FUNCTION_BLOCK TM_DO16 (* Extracted Composite Function Block Type *)
  (* Standard: 61499-2 *)
  (* Version 25/02/2026 *)
  PACKAGE Hidryco.HidrycoLib;
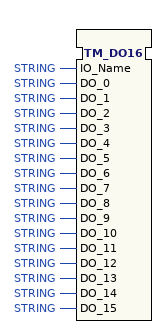
  VAR_INPUT
    IO_Name : STRING;
    DO_0 : STRING;
    DO_1 : STRING;
    DO_2 : STRING;
    DO_3 : STRING;
    DO_4 : STRING;
    DO_5 : STRING;
    DO_6 : STRING;
    DO_7 : STRING;
    DO_8 : STRING;
    DO_9 : STRING;
    DO_10 : STRING;
    DO_11 : STRING;
    DO_12 : STRING;
    DO_13 : STRING;
    DO_14 : STRING;
    DO_15 : STRING;
  END_VAR
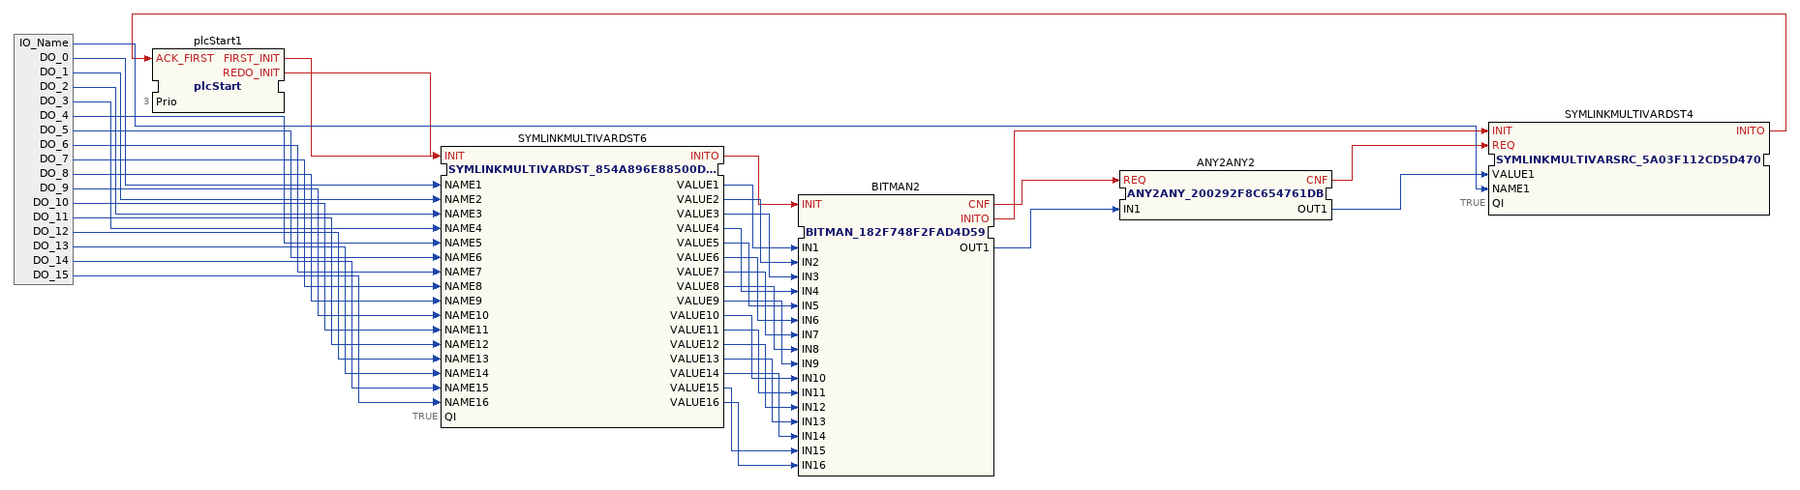
  FBS
    BITMAN2 : BITMAN_182F748F2FAD4D59; {SET_ATTRIBUTE(Configuration.GenericFBType.InterfaceParams, Runtime.Standard#CNTIN:=16;CNTOUT:=1;IN${CNTIN$}:BOOL,BOOL,BOOL,BOOL,BOOL,BOOL,BOOL,BOOL,BOOL,BOOL,BOOL,BOOL,BOOL,BOOL,BOOL,BOOL;OUT${CNTOUT$}:WORD)}
    ANY2ANY2 : ANY2ANY_200292F8C654761DB; {SET_ATTRIBUTE(Configuration.GenericFBType.InterfaceParams, Runtime.Standard#CNT:=1;IN${CNT$}:WORD;OUT${CNT$}:INT)}
    SYMLINKMULTIVARDST4 : SYMLINKMULTIVARSRC_5A03F112CD5D470(QI := TRUE); {SET_ATTRIBUTE(Configuration.GenericFBType.InterfaceParams, Runtime.System#I:=1;VALUE${I$}:INT)}
    SYMLINKMULTIVARDST6 : SYMLINKMULTIVARDST_854A896E88500D19(QI := TRUE); {SET_ATTRIBUTE(Configuration.GenericFBType.InterfaceParams, Runtime.System#I:=16;VALUE${I$}:BOOL,BOOL,BOOL,BOOL,BOOL,BOOL,BOOL,BOOL,BOOL,BOOL,BOOL,BOOL,BOOL,BOOL,BOOL,BOOL)}
    plcStart1 : plcStart(Prio := 3);
  END_FBS
  EVENT_CONNECTIONS
    BITMAN2.CNF TO ANY2ANY2.REQ;
    BITMAN2.INITO TO SYMLINKMULTIVARDST4.INIT;
    ANY2ANY2.CNF TO SYMLINKMULTIVARDST4.REQ;
    SYMLINKMULTIVARDST6.INITO TO BITMAN2.INIT;
    plcStart1.FIRST_INIT TO SYMLINKMULTIVARDST6.INIT;
    plcStart1.REDO_INIT TO SYMLINKMULTIVARDST6.INIT;
    SYMLINKMULTIVARDST4.INITO TO plcStart1.ACK_FIRST;
  END_CONNECTIONS
  DATA_CONNECTIONS
    BITMAN2.OUT1 TO ANY2ANY2.IN1;
    ANY2ANY2.OUT1 TO SYMLINKMULTIVARDST4.VALUE1;
    SYMLINKMULTIVARDST6.VALUE1 TO BITMAN2.IN1;
    SYMLINKMULTIVARDST6.VALUE2 TO BITMAN2.IN2;
    SYMLINKMULTIVARDST6.VALUE3 TO BITMAN2.IN3;
    SYMLINKMULTIVARDST6.VALUE4 TO BITMAN2.IN4;
    SYMLINKMULTIVARDST6.VALUE5 TO BITMAN2.IN5;
    SYMLINKMULTIVARDST6.VALUE6 TO BITMAN2.IN6;
    SYMLINKMULTIVARDST6.VALUE7 TO BITMAN2.IN7;
    SYMLINKMULTIVARDST6.VALUE8 TO BITMAN2.IN8;
    SYMLINKMULTIVARDST6.VALUE9 TO BITMAN2.IN9;
    SYMLINKMULTIVARDST6.VALUE10 TO BITMAN2.IN10;
    SYMLINKMULTIVARDST6.VALUE11 TO BITMAN2.IN11;
    SYMLINKMULTIVARDST6.VALUE12 TO BITMAN2.IN12;
    SYMLINKMULTIVARDST6.VALUE13 TO BITMAN2.IN13;
    SYMLINKMULTIVARDST6.VALUE14 TO BITMAN2.IN14;
    SYMLINKMULTIVARDST6.VALUE15 TO BITMAN2.IN15;
    SYMLINKMULTIVARDST6.VALUE16 TO BITMAN2.IN16;
    DO_0 TO SYMLINKMULTIVARDST6.NAME1;
    DO_1 TO SYMLINKMULTIVARDST6.NAME2;
    DO_2 TO SYMLINKMULTIVARDST6.NAME3;
    DO_3 TO SYMLINKMULTIVARDST6.NAME4;
    DO_4 TO SYMLINKMULTIVARDST6.NAME5;
    DO_5 TO SYMLINKMULTIVARDST6.NAME6;
    DO_6 TO SYMLINKMULTIVARDST6.NAME7;
    DO_7 TO SYMLINKMULTIVARDST6.NAME8;
    DO_8 TO SYMLINKMULTIVARDST6.NAME9;
    DO_9 TO SYMLINKMULTIVARDST6.NAME10;
    DO_10 TO SYMLINKMULTIVARDST6.NAME11;
    DO_11 TO SYMLINKMULTIVARDST6.NAME12;
    DO_12 TO SYMLINKMULTIVARDST6.NAME13;
    DO_13 TO SYMLINKMULTIVARDST6.NAME14;
    DO_14 TO SYMLINKMULTIVARDST6.NAME15;
    DO_15 TO SYMLINKMULTIVARDST6.NAME16;
    IO_Name TO SYMLINKMULTIVARDST4.NAME1;
  END_CONNECTIONS
END_FUNCTION_BLOCK
